PROGRAM MAIN
VAR
	PT1T2_Param		: S_PT1T2_Param;	// Parameter des Prozess
	PID_Param		: S_PID_Param;		// Parameter des Reglers
	Mode			: E_System_Mode := E_System_Mode.System_Init;	// Aktueller Modus
	T				: REAL;				// Abtastzeit
	PID_1			: FB_PID_Controller;// PID Regler Instanz
	PT1T2_1			: FB_PT1T2_Process; // PT1T2 System Instanz
	ref				: REAL;				// Referenzgroesse
	y_k				: REAL;				// Aktuelle Regelgroesse
	u_k				: REAL;				// Aktuelle Steuergroesse
END_VAR

CASE Mode OF
	E_System_Mode.System_Init:
		// set process variables
		PT1T2_Param.K 	:= 10;
		PT1T2_Param.T1 	:= 0.1;
		PT1T2_Param.T2 	:= 0.01;
		
		PID_Param.Kp 	:= 1/PT1T2_Param.K;
		PID_Param.Ti 	:= PT1T2_Param.T1;
		PID_Param.Td	:= PT1T2_Param.T2;
		PID_Param.N	 	:= 10;
		
		// initialize variables
		ref := 0;
		y_k := 0;
		u_k := 0;
		T := 0.001;
		
		// call process and controller to initialize them
		PT1T2_1(u := 0, Mode := Mode, Param := PT1T2_Param, T := T);
		PID_1(ref := 0, y := 0, Mode := Mode, Param := PID_Param, T := T);
		
		// change to run mode
		Mode := E_System_Mode.System_Run;
		
	E_System_Mode.System_Run:
		// call controller
		PID_1(ref := ref, y := y_k, Mode := Mode, Param := PID_Param, T := T);
		u_k := PID_1.u_k;
		
		// call process
		PT1T2_1(u := u_k, Mode := Mode, Param := PT1T2_Param, T := T);
		y_k := PT1T2_1.y;
		
	ELSE  // default assignment
	;
		
END_CASE

END_PROGRAM

(* stored: Version 1.1.0.1, ProductVersion 3.1.4024.9
   POU MAIN: Id {0ab64c77-f0ed-4726-a433-7ee9d5e73ed6}, SpecialFunc None *)
